(* IEC 61131-3 sources: Industry-PLC-LLM/data/PLCBEAD_repo/PLCBEAD_PLCEmbed-main/PLC-BEAD/Source/GEB/NEGX, 1 file *)

(* ---- NEGX.ST ---- *)
FUNCTION NEGX:REAL

	VAR_INPUT
		X :	REAL;
	END_VAR

	NEGX := -X;

END_FUNCTION

PROGRAM program0
	VAR
		_X : REAL;
		OUT : REAL;
	END_VAR

	OUT := NEGX(_X);
END_PROGRAM
